PROGRAM PRG_1_PlcTask
VAR
END_VAR

PRG_2_PMPS_PRE();

PRG_IM1K1_PPM();
PRG_IM2K1_PPM();
PRG_ST1K1_ZOS();
PRG_IM1K2_PPM();

PRG_3_PMPS_POST();
PRG_4_LOG();

END_PROGRAM

(* stored: Version 1.1.0.1, ProductVersion 3.1.4022.18
   POU PRG_1_PlcTask: Id {9c76104d-f8df-400f-b9a4-81d3480ca015}, SpecialFunc None *)
